// TIA Portal V17 export
// export: Created 2024-09-03T22:41:02.6909502Z, ExportSetting WithDefaults, DisplayName Totally Integrated Automation Portal, DisplayVersion V17 Update 7, DisplayName TIA Portal Openness, DisplayVersion V17 Update 7, DisplayName TIA Portal Version Control Interface, DisplayVersion V17, DisplayName SINAMICS Startdrive Advanced, DisplayVersion V17 SP2, DisplayName SINAMICS Startdrive G110M, G120, G120C, G120D, G120P, G115D, DisplayVersion V17 SP2, DisplayName SINAMICS Startdrive G130, G150, S120, S150, SINAMICS MV, S210, DisplayVersion V17 SP2, DisplayName STEP 7 Professional, DisplayVersion V17 Update 7, DisplayName STEP 7 Safety, DisplayVersion V17 Update 6, DisplayName WinCC Advanced / Unified PC, DisplayVersion V17 Update 7
TYPE "UDT_ProductionProgram"
// stored: IsFailsafeCompliant false
   STRUCT
      "Name" : String[50];
      CupformingParametersLeft { S7_SetPoint := 'True'} : "UDT_FittingParameters";
      CupformingParametersRight { S7_SetPoint := 'True'} : "UDT_FittingParameters";
      St1Insertion { S7_SetPoint := 'True'} : Array[1..20] of Bool;
      St1InsertionUsed : Array[1..20] of Bool;
      FaureciaNumber : String;
      FaureciaNumberStartChar : Int;
      FaureciaNumberLength : Int;
      MechanicalType : Int;
      Camera_program : Array[0..4] of USInt;
      Riveting_program_left : Array[0..2] of USInt;
      Riveting_program_right : Array[0..2] of USInt;
      Total_number_of_rivets_4 : Bool;
      NumberOfReadings : Int;
      Readings : Array[1..4] of "UDT_ProductionReadings";
      DMC : Array[1.."MaxRoundNumber", 1..10] of "DATA_DMC";
   END_STRUCT;
END_TYPE
